// SIMATIC S7-200 project (STEP 7-Micro/WIN), CPU 221 REL 01.10

SYMBOL_TABLE USER1
nut_1            I0.0
nut_2            I0.1
nut_3            I0.2
nut_4            I0.3
nut_5            I0.4
nut_6            I0.5
nut_7            I0.6
nut_8            I0.7
nut_9            I1.0
nut_10           I1.1
nut_11           I1.2
nut_12           I1.3
nut_13           I1.4
nut_14           I1.5
bong_1           Q0.0
bong_2           Q0.1
bong_3           Q0.2
bong_4           Q0.3
bong_5           Q0.4
bong_6           Q0.5
bong_7           Q0.6
bong_8           Q0.7
bong_9           Q1.0
bong_10          Q1.1
END_SYMBOL_TABLE

ORGANIZATION_BLOCK MAIN:OB1
TITLE=PROGRAM COMMENTS
BEGIN
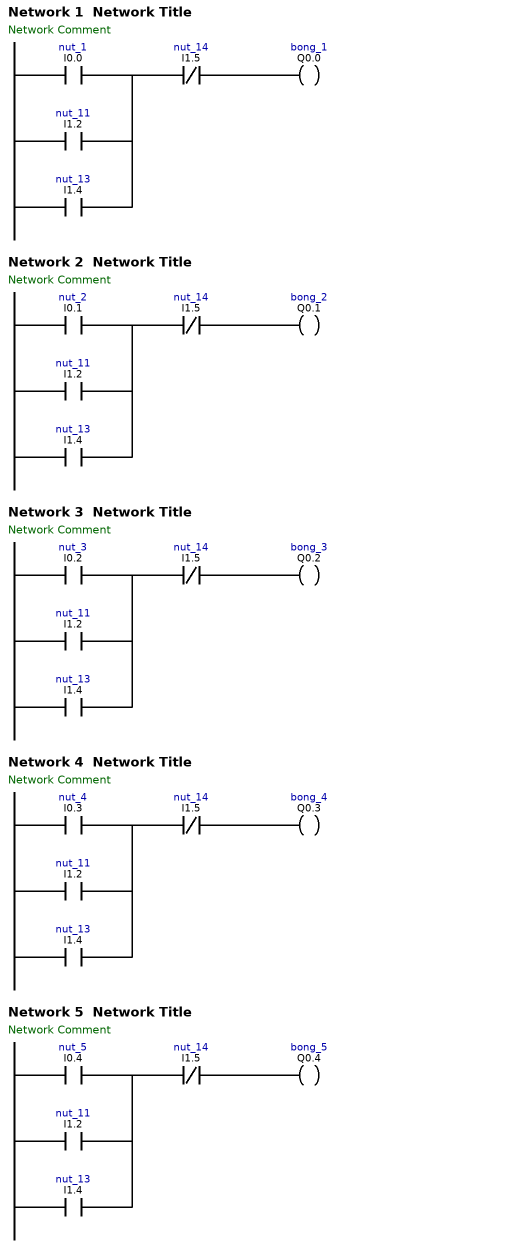
Network 1 // Network Title
// Network Comment
LD     nut_1:I0.0
O      nut_11:I1.2
O      nut_13:I1.4
AN     nut_14:I1.5
=      bong_1:Q0.0
Network 2 // Network Title
// Network Comment
// (network saved uncompiled; LAD cells follow)
// row 0: c0 -| |- nut_2:I0.1 v  c1 -|/|- nut_14:I1.5  c2 -( ) bong_2:Q0.1
// row 1: c0 -| |- nut_11:I1.2 ^v
// row 2: c0 -| |- nut_13:I1.4 ^
Network 3 // Network Title
// Network Comment
// (network saved uncompiled; LAD cells follow)
// row 0: c0 -| |- nut_3:I0.2 v  c1 -|/|- nut_14:I1.5  c2 -( ) bong_3:Q0.2
// row 1: c0 -| |- nut_11:I1.2 ^v
// row 2: c0 -| |- nut_13:I1.4 ^
Network 4 // Network Title
// Network Comment
// (network saved uncompiled; LAD cells follow)
// row 0: c0 -| |- nut_4:I0.3 v  c1 -|/|- nut_14:I1.5  c2 -( ) bong_4:Q0.3
// row 1: c0 -| |- nut_11:I1.2 ^v
// row 2: c0 -| |- nut_13:I1.4 ^
Network 5 // Network Title
// Network Comment
LD     nut_5:I0.4
O      nut_11:I1.2
O      nut_13:I1.4
AN     nut_14:I1.5
=      bong_5:Q0.4
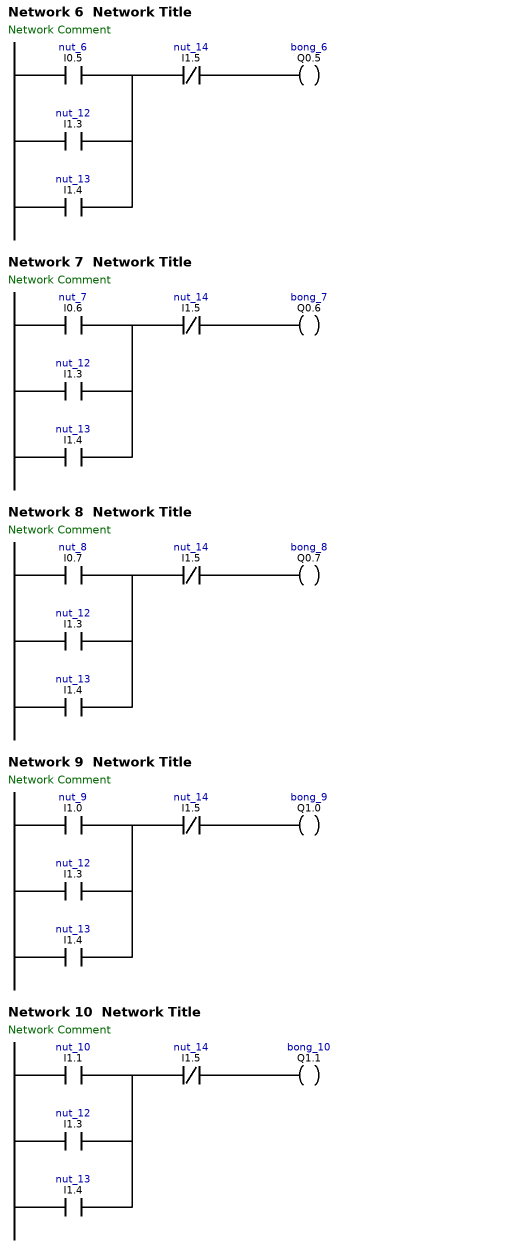
Network 6 // Network Title
// Network Comment
LD     nut_6:I0.5
O      nut_12:I1.3
O      nut_13:I1.4
AN     nut_14:I1.5
=      bong_6:Q0.5
Network 7 // Network Title
// Network Comment
LD     nut_7:I0.6
O      nut_12:I1.3
O      nut_13:I1.4
AN     nut_14:I1.5
=      bong_7:Q0.6
Network 8 // Network Title
// Network Comment
LD     nut_8:I0.7
O      nut_12:I1.3
O      nut_13:I1.4
AN     nut_14:I1.5
=      bong_8:Q0.7
Network 9 // Network Title
// Network Comment
LD     nut_9:I1.0
O      nut_12:I1.3
O      nut_13:I1.4
AN     nut_14:I1.5
=      bong_9:Q1.0
Network 10 // Network Title
// Network Comment
LD     nut_10:I1.1
O      nut_12:I1.3
O      nut_13:I1.4
AN     nut_14:I1.5
=      bong_10:Q1.1
END_ORGANIZATION_BLOCK
